RoboDK station: PDE4431_CW2.rdk

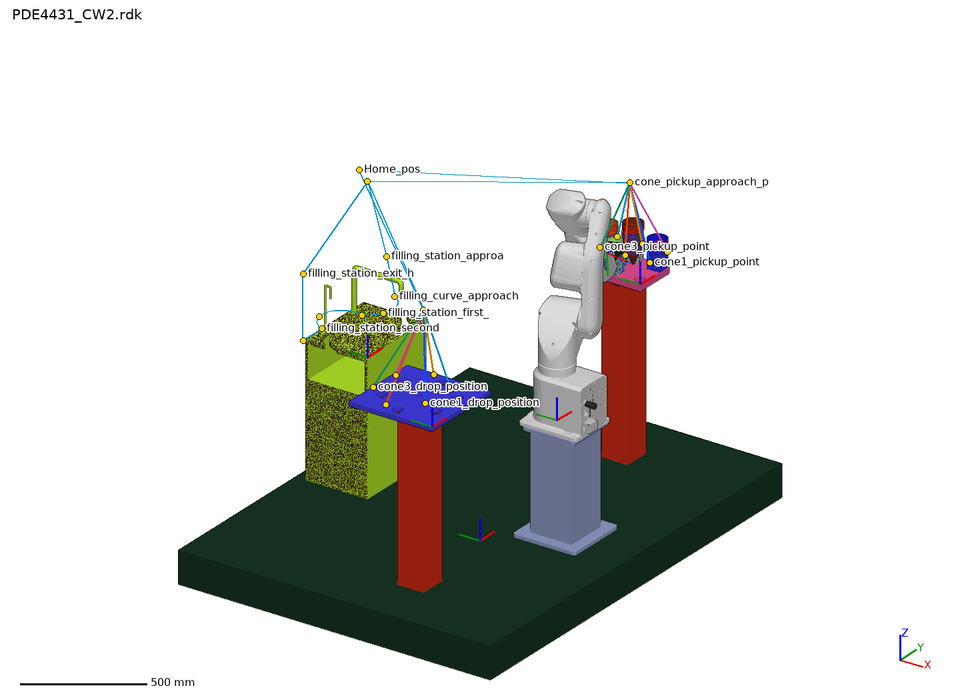
[picture v0: the station drawn from its stored meshes, robots at their saved joint values, targets as dots, program paths as lines]
Station pde4431_cw2_station (saved by RoboDK 5.8.0). Poses are relative to the parent item; angles as X-Y-Z fixed-axis rotations.
  - frame Base_Frame at (0, 0, 0) mm, rotated rx 0 ry 0 rz 90 deg
    - object PDE4431_CW2_2024 at (0, 0, 0) mm, size 2000 x 980 x 1500 mm, geometry from PDE4431_CW2_2024.STEP
    - object Pedestal_3 at (0, -410, 150) mm, rotated rx 90 ry 0 rz 0 deg, size 300 x 480 x 300 mm, geometry from Pedestal_3.STEP
    - frame Epson VT6 Base at (0, -370, 630) mm
      - robot Epson VT6: 6 axes, payload 6 kg, reach 920 mm, repeatability 0.1 mm, weight 40 kg
          modified DH rows (alpha deg, a mm, theta deg, d mm): 0, 0, 0, 412; -90, 100, -90, 0; 0, 420, 0, 0; -90, 0, 0, 400; 90, 0, 0, 0; -90, 0, 0, 80
          base shift (0, 0, 0) mm, rotated rx 0 ry 0 rz 90 deg
          joint limits [-170, -160, -51, -200, -125, -360] to [170, 65, 190, 200, 125, 360]; home [0, 0, 0, 0, 0, 0]; saved at [-72.982, -15.825, -37.748, -32.142, 60.244, 18.429]
        - frame RobotiQ 2F-85 Gripper (Mechanism) Base at (0, 0, 0) mm, rotated rx 0 ry 0 rz 90 deg
          - robot RobotiQ 2F-85 Gripper (Mechanism) (model RobotiQ 2F85): 1 axes, payload 5 kg
              joint limits [0] to [85]; home [85]; saved at [60]
          - object Cone1 at (4.06, -2.49, 139.78) mm, rotated rx 11.52 ry -79.28 rz 168.67 deg, size 84.9 x 182 x 85 mm, geometry from Cone-Part.STEP
        - tool Tool 1, TCP at (0, 0, 200) mm
      - target target_gripper_close (Cartesian target) at (0, 683, 832) mm, rotated rx -90 ry 0 rz 0 deg; joints [0, 0, 0, 0, 0, 0] of RobotiQ 2F-85 Gripper (Mechanism)
      - target target_gripper_grip (Cartesian target) at (0, 683.92, 832) mm, rotated rx -90 ry 0 rz 0 deg; joints [60, 0, 0, 0, 0, 0] of RobotiQ 2F-85 Gripper (Mechanism)
      - target target_gripper_open (Cartesian target) at (0, 683.92, 832) mm, rotated rx -90 ry 0 rz 0 deg; joints [85, 0, 0, 0, 0, 0] of RobotiQ 2F-85 Gripper (Mechanism)
    - frame feed_Frame at (600, -350, 980) mm
      - object Cone6 at (160, 270, 50) mm, rotated rx 90 ry 0 rz 0 deg, size 84.9 x 182 x 85 mm, geometry from Cone-Part.STEP
      - object Cone3 at (40, 270, 50) mm, rotated rx 90 ry 0 rz 0 deg, size 84.9 x 182 x 85 mm, geometry from Cone-Part.STEP
      - object Cone4 at (160, 30, 50) mm, rotated rx 90 ry 0 rz 0 deg, size 84.9 x 182 x 85 mm, geometry from Cone-Part.STEP
      - object Cone5 at (160, 150, 50) mm, rotated rx 90 ry 0 rz 0 deg, size 84.9 x 182 x 85 mm, geometry from Cone-Part.STEP
      - object Cone2 at (40, 150, 50) mm, rotated rx 90 ry 0 rz 0 deg, size 84.9 x 182 x 85 mm, geometry from Cone-Part.STEP
    - frame drop_Frame at (-900, -400, 970) mm
    - frame filling_station_frame at (-200, 400, 770) mm
    - target Home_pos (Cartesian target) at (0, 580, 1462) mm, rotated rx 0 ry -90 rz -90 deg; joints [0, 0, 0, 0, 0, 0] of Epson VT6
    - target cone_pickup_approach_pt (Cartesian target) at (721.78, -213.9, 1339.75) mm, rotated rx 0 ry -87.87 rz 169.49 deg; joints [-65.121, -2.034, -17.294, -62.232, 40.847, 56.673] of Epson VT6
    - target cone1_pickup_point (Cartesian target) at (700, -327, 1029.75) mm, rotated rx 0 ry -87.87 rz 169.49 deg; joints [-100.136, -30.937, -42.249, -0.386, 75.317, 0.112] of Epson VT6
    - target cone2_pickup_point (Cartesian target) at (700, -207, 1029.75) mm, rotated rx 0 ry -87.87 rz 169.49 deg; joints [-63.263, -33.451, -35.412, -38.685, 75.393, 13.035] of Epson VT6
    - target cone3_pickup_point (Cartesian target) at (700, -87, 1029.75) mm, rotated rx 0 ry -87.87 rz 169.49 deg; joints [-51.826, -37.648, -24.976, -51.223, 74.313, 21.022] of Epson VT6
    - target cone4_pickup_point (Cartesian target) at (820, -327, 1029.75) mm, rotated rx 0 ry -87.87 rz 169.49 deg; joints [-80.208, -38.521, -22.897, -22.41, 65.434, 10.516] of Epson VT6
    - target cone5_pickup_point (Cartesian target) at (820, -207, 1029.75) mm, rotated rx 0 ry -87.87 rz 169.49 deg; joints [-68.554, -40.892, -17.36, -35.534, 65.511, 17.819] of Epson VT6
    - target cone6_pickup_point (Cartesian target) at (820, -87, 1029.75) mm, rotated rx 0 ry -87.87 rz 169.49 deg; joints [-58.49, -45.138, -7.736, -47.435, 65.263, 26.413] of Epson VT6
    - target filling_station_approach_point (Cartesian target) at (213.98, 599.85, 991.54) mm, rotated rx 59.3 ry -85.13 rz -160.71 deg; joints [-14.49, -49.38, -7.77, 183.67, -59.69, 0] of Epson VT6
    - target filling_curve_approach (Cartesian target) at (227.21, 567.56, 819.75) mm, rotated rx 0 ry -87.87 rz -110.51 deg; joints [-12.239, -69.096, -3.898, 171.453, -75.305, -177.507] of Epson VT6
    - target filling_station_first_curve (Cartesian target) at (77.21, 517.56, 819.75) mm, rotated rx 0 ry -87.87 rz -110.51 deg; joints [2.618, -66.684, -27.579, -10, 96.048, -1.682] of Epson VT6
    - target filling_station_first_curve_end (Cartesian target) at (17.21, 577.56, 819.75) mm, rotated rx 0 ry -87.87 rz -110.51 deg; joints [8.911, -66.759, -18.096, -29.426, 87.647, 2.527] of Epson VT6
    - target filling_station_second_curve_mid (Cartesian target) at (-92.79, 707.56, 819.75) mm, rotated rx 0 ry -87.87 rz -110.51 deg; joints [16.469, -72.262, 7.901, -39.248, 71.825, 15.899] of Epson VT6
    - target filling_station_second_curve_end (Cartesian target) at (-172.79, 637.56, 819.75) mm, rotated rx 0 ry -87.87 rz -110.51 deg; joints [25.202, -70.27, 0.863, -47.034, 77.84, 14.925] of Epson VT6
    - target filling_station_exit (Cartesian target) at (-302.79, 637.56, 819.75) mm, rotated rx 0 ry -87.87 rz -110.51 deg; joints [34.857, -74.078, 13.655, -58.077, 75.641, 24.786] of Epson VT6
    - target filling_station_exit_high (Cartesian target) at (-302.79, 637.56, 1109.75) mm, rotated rx 0 ry -87.87 rz -110.51 deg; joints [34.857, -43.267, 4.863, -65.085, 65.042, 45.333] of Epson VT6
    - target drop_station_approach_high (Cartesian target) at (-695, -215.04, 1350) mm, rotated rx 39.86 ry -87.87 rz -52.23 deg; joints [77.29, 6.882, -23.887, 1.118, 18.645, 0.299] of Epson VT6
    - target safe_point (Cartesian target) at (0, 540, 1422) mm, rotated rx 0 ry -90 rz -90 deg; joints [0, 5.214, -10.703, 0, 5.489, 0] of Epson VT6
    - target cone1_drop_position (Cartesian target) at (-825, -315.04, 1020) mm, rotated rx 39.86 ry -87.87 rz -52.23 deg; joints [90.51, -39.389, -23.048, 165.765, -64.812, -172.096] of Epson VT6
    - target cone2_drop_position (Cartesian target) at (-925, -195.04, 1020) mm, rotated rx 39.86 ry -87.87 rz -52.23 deg; joints [79.983, -47.833, -3.415, 177.073, -52.923, -176.799] of Epson VT6
    - target cone3_drop_position (Cartesian target) at (-825, -65.04, 1020) mm, rotated rx 39.86 ry -87.87 rz -52.23 deg; joints [73.338, -41.087, -18.955, 184.891, -61.773, -181.073] of Epson VT6
    - target cone4_drop_position (Cartesian target) at (-685, -75.04, 1020) mm, rotated rx 39.86 ry -87.87 rz -32.23 deg; joints [50.819, -37.668, -27.311, 49.086, 74.731, -17.28] of Epson VT6
    - target cone5_drop_position (Cartesian target) at (-595, -195.04, 1020) mm, rotated rx 39.86 ry -87.87 rz -32.24 deg; joints [56.251, -30.054, -49.63, 41.663, 83.906, -5.471] of Epson VT6
    - target cone6_drop_position (Cartesian target) at (-665, -325.04, 1020) mm, rotated rx 39.86 ry -87.87 rz -52.24 deg; joints [92.181, -30.441, -48.156, -14.729, 80.603, 4.251] of Epson VT6
  - program replace_all_cones (1 instructions, listed below)
  - program gripper_open (2 instructions, listed below)
  - program gripper_grip (2 instructions, listed below)
  - program gripper_close (2 instructions, listed below)
  - program move_cone_1 (24 instructions, listed below)
  - program attach_to_tool (1 instructions, listed below)
  - program detach_from_tool (1 instructions, listed below)
  - Python program MainProrgram (listed below)
  - program move_cone_2 (24 instructions, listed below)
  - program move_cone_3 (24 instructions, listed below)
  - program move_cone_4 (24 instructions, listed below)
  - program move_cone_5 (24 instructions, listed below)
  - program move_cone_6 (24 instructions, listed below)
  - program MasterProgram (7 instructions, listed below)
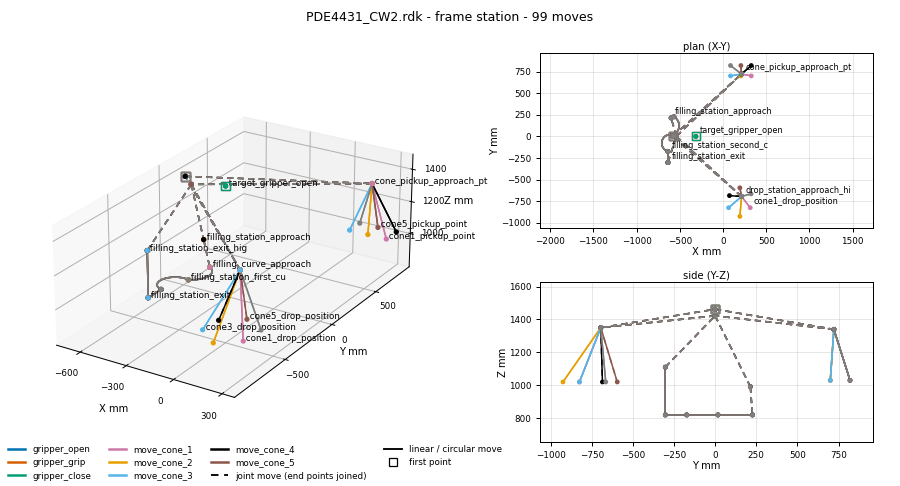
[picture p0: tool path of PDE4431_CW2.rdk in frame station, 99 of 99 moves have a stored position in this frame; points joined in program order, loops and branches not executed]

--- program replace_all_cones (robot Epson VT6) ---
  Replace objects

--- program gripper_open (robot RobotiQ 2F-85 Gripper (Mechanism)) ---
  Set Ref.: Epson VT6 Base
  MoveJ (target_gripper_open)

--- program gripper_grip (robot RobotiQ 2F-85 Gripper (Mechanism)) ---
  Set Ref.: Epson VT6 Base
  MoveJ (target_gripper_grip)

--- program gripper_close (robot RobotiQ 2F-85 Gripper (Mechanism)) ---
  Set Ref.: Epson VT6 Base
  MoveJ (target_gripper_close)

--- program move_cone_1 (robot Epson VT6) ---
  Set Ref.: Base_Frame
  Set Tool: Tool 1
  MoveJ (Home_pos)
  Call gripper_open
  MoveJ (cone_pickup_approach_pt)
  MoveL (cone1_pickup_point)
  Call gripper_grip
  Attach to Tool 1
  MoveL (cone_pickup_approach_pt)
  MoveJ (safe_point)
  MoveJ (filling_station_approach_point)
  MoveJ (filling_curve_approach)
  MoveC (filling_station_first_curve, filling_station_first_curve_end)
  MoveC (filling_station_second_curve_mid, filling_station_second_curve_end)
  MoveL (filling_station_exit)
  MoveL (filling_station_exit_high)
  MoveJ (safe_point)
  MoveJ (drop_station_approach_high)
  MoveL (cone1_drop_position)
  Call gripper_open
  Detach from Tool 1
  MoveL (drop_station_approach_high)
  Call gripper_close
  MoveJ (Home_pos)

--- program attach_to_tool (robot Epson VT6) ---
  Attach to Tool 1

--- program detach_from_tool (robot Epson VT6) ---
  Detach from Tool 1

--- Python program MainProrgram ---
# Type help("robodk.robolink") or help("robodk.robomath") for more information
# Press F5 to run the script
# Documentation: https://robodk.com/doc/en/RoboDK-API.html
# Reference:     https://robodk.com/doc/en/PythonAPI/robodk.html
# Note: It is not required to keep a copy of this file, your Python script is saved with your RDK project

# You can also use the new version of the API:
from robodk import robolink    # RoboDK API
from robodk import robomath    # Robot toolbox
import time
from robodk import *      # RoboDK API
from robolink import *    # Robot toolbox

RDK = robolink.Robolink()
coursework_bot = RDK.Item('Epson VT6')
coursework_bot.setSpeed(100)

# variables and location teaching start

# programs

gripper_open_function = RDK.Item('gripper_open', itemtype=ITEM_TYPE_PROGRAM)
gripper_close_function = RDK.Item('gripper_close', itemtype=ITEM_TYPE_PROGRAM)
gripper_grip_function = RDK.Item('gripper_grip', itemtype=ITEM_TYPE_PROGRAM)
attach_to_tool = RDK.Item('attach_to_tool', itemtype=ITEM_TYPE_PROGRAM)
detach_from_tool = RDK.Item('detach_from_tool', itemtype=ITEM_TYPE_PROGRAM)
replace_all_cones = RDK.Item('replace_all_cones', itemtype=ITEM_TYPE_PROGRAM)

# frames for pickup and drop
feed_frame = RDK.Item('feed_frame')
outfeed_frame = RDK.Item('drop_frame')
gripper_tool = coursework_bot.Childs()[0]

# Cone pick up station locations
cone1_pickup_loc = RDK.Item('cone1_pickup_point')
cone2_pickup_loc = cone1_pickup_loc.Pose() * transl(0,-120, 0)
cone3_pickup_loc = cone1_pickup_loc.Pose() * transl(0,-240, 0)
cone4_pickup_loc = cone1_pickup_loc.Pose() * transl(0,0, 120)
cone5_pickup_loc = cone1_pickup_loc.Pose() * transl(0,-120, 120)
cone6_pickup_loc = cone1_pickup_loc.Pose() * transl(0,-240, 120)

# cone drop locations
cone1_drop_loc = RDK.Item('cone1_drop_position', itemtype=ITEM_TYPE_TARGET)
cone2_drop_loc = RDK.Item('cone2_drop_position', itemtype=ITEM_TYPE_TARGET)
cone3_drop_loc = RDK.Item('cone3_drop_position', itemtype=ITEM_TYPE_TARGET)
cone4_drop_loc = RDK.Item('cone4_drop_position', itemtype=ITEM_TYPE_TARGET)
cone5_drop_loc = RDK.Item('cone5_drop_position', itemtype=ITEM_TYPE_TARGET)
cone6_drop_loc = RDK.Item('cone6_drop_position', itemtype=ITEM_TYPE_TARGET)


# points for movement
home_pos = RDK.Item('Home_pos')
cone_pickup_approach_point = RDK.Item('cone_pickup_approach_pt')
safe_point = RDK.Item('safe_point')
filling_station_approach_point = RDK.Item('filling_station_approach_point')
filling_curve_approach = RDK.Item('filling_curve_approach')
filling_station_exit = RDK.Item('filling_station_exit')
filling_station_exit_high = RDK.Item('filling_station_exit_high')
drop_station_approach_high = RDK.Item('drop_station_approach_high')

# curve points for filling station
filling_station_first_curve = RDK.Item('filling_station_first_curve')
filling_station_first_curve_end = RDK.Item('filling_station_first_curve_end')
filling_station_second_curve_mid = RDK.Item('filling_station_second_curve_mid')
filling_station_second_curve_end = RDK.Item('filling_station_second_curve_end')

# variables and location teaching end

# main execution starts here

pickup_positions = [cone1_pickup_loc, cone2_pickup_loc, cone3_pickup_loc, cone4_pickup_loc, cone5_pickup_loc, cone6_pickup_loc]
drop_locations = [cone1_drop_loc, cone2_drop_loc, cone3_drop_loc, cone4_drop_loc, cone5_drop_loc, cone6_drop_loc]
cone_list = ['Cone1', 'Cone2', 'Cone3', 'Cone4', 'Cone5', 'Cone6']
replace_all_cones.RunCode()
for i in range(6):
    coursework_bot.MoveJ(home_pos)
    gripper_open_function.RunCode()
    coursework_bot.MoveJ(cone_pickup_approach_point)
    coursework_bot.MoveL(pickup_positions[i])
    gripper_grip_function.RunCode()
    # attach_to_tool.RunCode()
    attach_object = RDK.Item(cone_list[i])
    curr_pose = attach_object.PoseAbs()
    attach_object.setParent(gripper_tool)
    attach_object.setPoseAbs(curr_pose)
    coursework_bot.MoveL(cone_pickup_approach_point)
    coursework_bot.MoveJ(safe_point)
    coursework_bot.MoveJ(filling_station_approach_point)
    coursework_bot.MoveJ(filling_curve_approach)
    coursework_bot.MoveC(filling_station_first_curve, filling_station_first_curve_end)
    coursework_bot.MoveC(filling_station_second_curve_mid, filling_station_second_curve_end)
    coursework_bot.MoveL(filling_station_exit)
    coursework_bot.MoveL(filling_station_exit_high)
    coursework_bot.MoveJ(safe_point)
    coursework_bot.MoveJ(drop_station_approach_high)
    # if i == 4 or i == 5:
    #     coursework_bot.MoveJ(drop_locations[i])
    # else:
    coursework_bot.MoveJ(drop_locations[i])
    detach_from_tool.RunCode()
    print(cone_list[i])
    detach_object = RDK.Item(cone_list[i])
    drop_pose = detach_object.PoseAbs()
    print(drop_pose)
    detach_object.setParent(outfeed_frame)
    detach_object.setPoseAbs(drop_pose)
    gripper_open_function.RunCode()
    coursework_bot.MoveJ(drop_station_approach_high)
    gripper_close_function.RunCode()
    coursework_bot.MoveJ(home_pos)

--- program move_cone_2 (robot Epson VT6) ---
  Set Ref.: Base_Frame
  Set Tool: Tool 1
  MoveJ (Home_pos)
  Call gripper_open
  MoveJ (cone_pickup_approach_pt)
  MoveL (cone2_pickup_point)
  Call gripper_grip
  Attach to Tool 1
  MoveL (cone_pickup_approach_pt)
  MoveJ (safe_point)
  MoveJ (filling_station_approach_point)
  MoveJ (filling_curve_approach)
  MoveC (filling_station_first_curve, filling_station_first_curve_end)
  MoveC (filling_station_second_curve_mid, filling_station_second_curve_end)
  MoveL (filling_station_exit)
  MoveL (filling_station_exit_high)
  MoveJ (safe_point)
  MoveJ (drop_station_approach_high)
  MoveL (cone2_drop_position)
  Call gripper_open
  Detach from Tool 1
  MoveL (drop_station_approach_high)
  Call gripper_close
  MoveJ (Home_pos)

--- program move_cone_3 (robot Epson VT6) ---
  Set Ref.: Base_Frame
  Set Tool: Tool 1
  MoveJ (Home_pos)
  Call gripper_open
  MoveJ (cone_pickup_approach_pt)
  MoveL (cone3_pickup_point)
  Call gripper_grip
  Attach to Tool 1
  MoveL (cone_pickup_approach_pt)
  MoveJ (safe_point)
  MoveJ (filling_station_approach_point)
  MoveJ (filling_curve_approach)
  MoveC (filling_station_first_curve, filling_station_first_curve_end)
  MoveC (filling_station_second_curve_mid, filling_station_second_curve_end)
  MoveL (filling_station_exit)
  MoveL (filling_station_exit_high)
  MoveJ (safe_point)
  MoveJ (drop_station_approach_high)
  MoveL (cone3_drop_position)
  Call gripper_open
  Detach from Tool 1
  MoveL (drop_station_approach_high)
  Call gripper_close
  MoveJ (Home_pos)

--- program move_cone_4 (robot Epson VT6) ---
  Set Ref.: Base_Frame
  Set Tool: Tool 1
  MoveJ (Home_pos)
  Call gripper_open
  MoveJ (cone_pickup_approach_pt)
  MoveL (cone4_pickup_point)
  Call gripper_grip
  Attach to Tool 1
  MoveL (cone_pickup_approach_pt)
  MoveJ (safe_point)
  MoveJ (filling_station_approach_point)
  MoveJ (filling_curve_approach)
  MoveC (filling_station_first_curve, filling_station_first_curve_end)
  MoveC (filling_station_second_curve_mid, filling_station_second_curve_end)
  MoveL (filling_station_exit)
  MoveL (filling_station_exit_high)
  MoveJ (safe_point)
  MoveJ (drop_station_approach_high)
  MoveJ (cone4_drop_position)
  Call gripper_open
  Detach from Tool 1
  MoveL (drop_station_approach_high)
  Call gripper_close
  MoveJ (Home_pos)

--- program move_cone_5 (robot Epson VT6) ---
  Set Ref.: Base_Frame
  Set Tool: Tool 1
  MoveJ (Home_pos)
  Call gripper_open
  MoveJ (cone_pickup_approach_pt)
  MoveL (cone5_pickup_point)
  Call gripper_grip
  Attach to Tool 1
  MoveL (cone_pickup_approach_pt)
  MoveJ (safe_point)
  MoveJ (filling_station_approach_point)
  MoveJ (filling_curve_approach)
  MoveC (filling_station_first_curve, filling_station_first_curve_end)
  MoveC (filling_station_second_curve_mid, filling_station_second_curve_end)
  MoveL (filling_station_exit)
  MoveL (filling_station_exit_high)
  MoveJ (safe_point)
  MoveJ (drop_station_approach_high)
  MoveJ (cone5_drop_position)
  Call gripper_open
  Detach from Tool 1
  MoveL (drop_station_approach_high)
  Call gripper_close
  MoveJ (Home_pos)

--- program move_cone_6 (robot Epson VT6) ---
  Set Ref.: Base_Frame
  Set Tool: Tool 1
  MoveJ (Home_pos)
  Call gripper_open
  MoveJ (cone_pickup_approach_pt)
  MoveL (cone6_pickup_point)
  Call gripper_grip
  Attach to Tool 1
  MoveL (cone_pickup_approach_pt)
  MoveJ (safe_point)
  MoveJ (filling_station_approach_point)
  MoveJ (filling_curve_approach)
  MoveC (filling_station_first_curve, filling_station_first_curve_end)
  MoveC (filling_station_second_curve_mid, filling_station_second_curve_end)
  MoveL (filling_station_exit)
  MoveL (filling_station_exit_high)
  MoveJ (safe_point)
  MoveJ (drop_station_approach_high)
  MoveL (cone6_drop_position)
  Call gripper_open
  Detach from Tool 1
  MoveL (drop_station_approach_high)
  Call gripper_close
  MoveJ (Home_pos)

--- program MasterProgram (robot Epson VT6) ---
  Call replace_all_cones
  Call move_cone_1
  Call move_cone_2
  Call move_cone_3
  Call move_cone_4
  Call move_cone_5
  Call move_cone_6
